// Mitsubishi GX Works2 project: De04   PLC: FX2N/FX2NC

PROGRAM MAIN
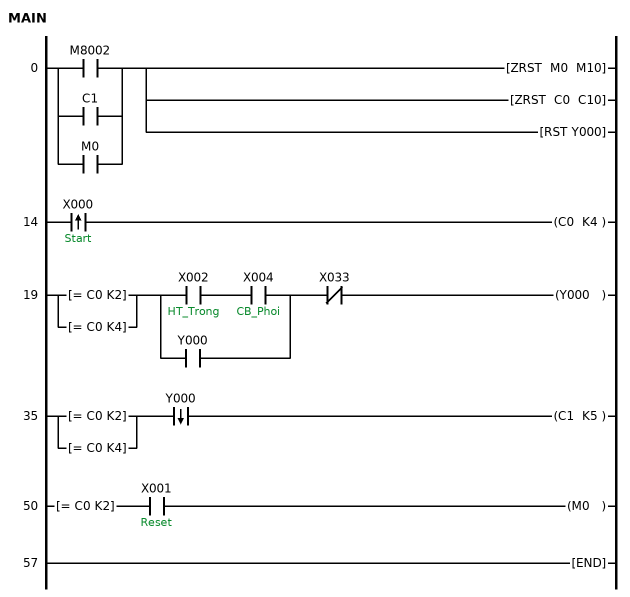
0     LD      M8002
      OR      C1
      OR      M0
      ZRST    M0 M10
      ZRST    C0 C10
      RST     Y000
14    LDP     X000  ; Start
      OUT     C0 K4
19    LD=     C0 K2
      OR=     C0 K4
      LD      X002  ; HT_Trong
      AND     X004  ; CB_Phoi
      OR      Y000
      ANB
      ANI     X033
      OUT     Y000
35    LD=     C0 K2
      OR=     C0 K4
      ANDF    Y000
      OUT     C1 K5
50    LD=     C0 K2
      AND     X001  ; Reset
      OUT     M0
57    END
END_PROGRAM

// device comments not shown above
X003  ; HT_Ngoai
